not-CDATA

(* stored: DUT X: Id {x} *)
